// TIA Portal V20 export
DATA_BLOCK "DB_AnalogOutputs"   // DB2113
// stored: AutoNumber false, InstanceOfName FB_AnalogOutputs, InstanceOfType FB
"FB_AnalogOutputs"
   // VAR
   //    sNozzleOverpressureSetPoint { S7_SetPoint := 'True'} : "FB_AnalogOutput";
   //    sFreeQW482 { S7_SetPoint := 'True'} : "FB_AnalogOutput";
   //    sVentilatorSetPoint { S7_SetPoint := 'True'} : "FB_AnalogOutput";
   //    sPropValveClimSetPoint { S7_SetPoint := 'True'} : "FB_AnalogOutput";
   // END_VAR
BEGIN
END_DATA_BLOCK
